# EPICS autosave request: SPApp/Db/VindumPumpN_settings.req
$(P)$(PUMP)SetPressure
$(P)$(PUMP)PressureHOPR
$(P)$(PUMP)PressureLOPR
$(P)$(PUMP)PressureTweak
$(P)$(PUMP)SafetyPressure
$(P)$(PUMP)SetFlowRate
$(P)$(PUMP)SetVolume
$(P)$(PUMP)FlowRateTweak
$(P)$(PUMP)PumpMode
$(P)$(PUMP)AutofillMode
$(P)$(PUMP)VolumeMode
$(P)$(PUMP)Direction
$(P)$(PUMP)DeliverValve
$(P)$(PUMP)FillValve
$(P)$(PUMP)Description
